// TwinCAT 3 PLC project Untitled1
// ProgramVersion: 3.1.4026.11
// libraries:
//   Tc2_Standard, * (Beckhoff Automation GmbH)
//   Tc2_System, * (Beckhoff Automation GmbH)
//   Tc2_Utilities, * (Beckhoff Automation GmbH)
// project tree:
//   CommandInvoker/ FB_CommandInvoker.TcPOU, I_CommandInvoker.TcIO
//   Command/AxisCommandExample/ FB_AxisCommandFactory.TcPOU (not stored), FB_AxisMoveCommand.TcPOU
//   Command/FlowCommands/ FB_CompositeCommand.TcPOU, FB_FlowCommandFactory.TcPOU, FB_WaitCommand.TcPOU, FB_WaitForConditionCommand.TcPOU
//   Command/ I_Command.TcIO
//   Command/ValveCommandExample/ FB_ValveCommandFactory.TcPOU (not stored), FB_ValveMoveCommand.TcPOU
//   Components/Axis/ FB_Axis.TcPOU (not stored), I_Axis.TcIO (not stored)
//   Components/Valve/ E_ValvePosition.TcDUT, FB_Valve.TcPOU, I_Valve.TcIO
//   General/Datatypes/ Integer.TcDUT (not stored), Positive.TcDUT (not stored), Number.TcDUT
//   General/ FB_Base.TcPOU, F_Log.TcPOU
//   InplaceStringBuilder/ FB_StringBuilder.TcPOU, F_BuildString.TcPOU
//   / MAIN.TcPOU, PlcTask.TcTTO
//   Progress/ E_ProgressStatus.TcDUT, FB_Progress.TcPOU, I_Progress.TcIO
//   Values/Binding/ Value.TcPOU, FB_BoolBindingReadOnly.TcPOU, I_BoolBindable.TcIO (not stored), NotValue.TcPOU
//   Values/BooleanExpression/ Or2.TcPOU, And3.TcPOU, Or3.TcPOU, And4.TcPOU, Or4.TcPOU, And5.TcPOU, Or5.TcPOU, E_BooleanOperator.TcDUT, FB_BooleanExpression.TcPOU, And2.TcPOU
//   Values/ BoolValues.TcGVL, FB_TrueBoolValue.TcPOU, FB_FalseBoolValue.TcPOU, I_BoolValue.TcIO
// real-time tasks:
//   TASK PlcTask: cycle T#10ms, priority 20, ADS port 350

CONFIGURATION Untitled1
    RESOURCE PLC ON TwinCAT3
        TASK PlcTask(INTERVAL := T#10ms, PRIORITY := 20);
        PROGRAM MAIN WITH PlcTask : MAIN;
    END_RESOURCE
END_CONFIGURATION

// ---- Components/Valve/E_ValvePosition.TcDUT
{attribute 'qualified_only'}
{attribute 'strict'}
{attribute 'to_string'}
TYPE E_ValvePosition :
(
	Home,
	Work
);
END_TYPE

// ---- General/Datatypes/Number.TcDUT
TYPE Number : LREAL; END_TYPE

// ---- Progress/E_ProgressStatus.TcDUT
{attribute 'qualified_only'}
{attribute 'strict'}
{attribute 'to_string'}
TYPE E_ProgressStatus :
(
	Idle,
	Running,
	Paused,
	Completed,
	Error
);
END_TYPE

// ---- Values/BooleanExpression/E_BooleanOperator.TcDUT
{attribute 'qualified_only'}
{attribute 'strict'}
{attribute 'to_string'}
TYPE E_BooleanOperator :
(
	ANDop,
	ORop,
	XORop
);
END_TYPE

// ---- Values/BoolValues.TcGVL
{attribute 'qualified_only'}
VAR_GLOBAL CONSTANT
	FalseValue : FB_FalseBoolValue := ();
	TrueValue : FB_TrueBoolValue := ();
END_VAR

// ---- CommandInvoker/I_CommandInvoker.TcIO
INTERFACE I_CommandInvoker

METHOD AddCommand : BOOL
VAR_INPUT
	command : I_Command;
END_VAR
END_METHOD

METHOD ClearCommands
VAR
END_VAR
END_METHOD

{attribute 'monitoring' := 'call'}
PROPERTY CommandCount : INT
GET
END_GET
END_PROPERTY

METHOD Cyclic
VAR_INPUT
END_VAR
END_METHOD

{attribute 'monitoring' := 'call'}
PROPERTY InvokeIndex : INT
GET
END_GET
END_PROPERTY

METHOD Pause
VAR_INPUT
END_VAR
END_METHOD

{attribute 'monitoring' := 'call'}
PROPERTY PauseRequest : BOOL
GET
END_GET
END_PROPERTY

{attribute 'monitoring' := 'call'}
PROPERTY ProgressPercent : REAL
GET
END_GET
END_PROPERTY

{attribute 'monitoring' := 'call'}
PROPERTY ProgressState : E_ProgressStatus
GET
END_GET
END_PROPERTY

METHOD Reset
VAR_INPUT
END_VAR
END_METHOD

METHOD ResetCommands : BOOL
VAR
END_VAR
END_METHOD

METHOD Start
VAR_INPUT
END_VAR
END_METHOD

{attribute 'monitoring' := 'call'}
PROPERTY StepMode : BOOL
GET
END_GET
SET
END_SET
END_PROPERTY

END_INTERFACE

// ---- Command/I_Command.TcIO
INTERFACE I_Command EXTENDS __SYSTEM.IQueryInterface

{attribute 'monitoring' := 'call'}
PROPERTY Description : STRING
GET
END_GET
END_PROPERTY

METHOD Execute : E_ProgressStatus
VAR_INPUT
END_VAR
END_METHOD

METHOD Reset
VAR_INPUT
END_VAR
END_METHOD

END_INTERFACE

// ---- Components/Valve/I_Valve.TcIO
INTERFACE I_Valve

METHOD MoveToHome : BOOL
VAR_INPUT
END_VAR
END_METHOD

METHOD MoveToWork : BOOL
VAR_INPUT
END_VAR
END_METHOD

END_INTERFACE

// ---- Progress/I_Progress.TcIO
INTERFACE I_Progress

{attribute 'monitoring' := 'call'}
PROPERTY CompletedCount : INT
GET
END_GET
SET
END_SET
END_PROPERTY

{attribute 'monitoring' := 'call'}
PROPERTY Count : INT
GET
END_GET
SET
END_SET
END_PROPERTY

{attribute 'monitoring' := 'call'}
PROPERTY Percent : REAL
GET
END_GET
END_PROPERTY

{attribute 'monitoring' := 'call'}
PROPERTY PercentString : STRING
GET
END_GET
END_PROPERTY

{attribute 'monitoring' := 'call'}
PROPERTY UnitProgress : REAL // Progress 0..1
GET
END_GET
END_PROPERTY

END_INTERFACE

// ---- Values/I_BoolValue.TcIO
INTERFACE I_BoolValue EXTENDS __SYSTEM.IQueryInterface

{attribute 'monitoring' := 'call'}
PROPERTY Value : BOOL
GET
END_GET
END_PROPERTY

END_INTERFACE

// ---- MAIN.TcPOU
PROGRAM MAIN
VAR
	valve : FB_Valve;
	axis : FB_Axis;
	valveFactory : FB_ValveCommandFactory;
	axisFactory : FB_AxisCommandFactory;
	flowFactory : FB_FlowCommandFactory;
	
	invoker : FB_CommandInvoker<20>;
	subsequence : FB_CommandInvoker<10>;
	
	start : BOOL;
	create : BOOL;
	
	pauseIndex : INT := -1;
	
	test : BOOL;
	test2 : BOOL;
	test3 : BOOL;
	test4 : BOOL;
	
	val : I_BoolValue;
END_VAR

IF create THEN
	create := FALSE;
	
	subsequence.AddCommand(valveFactory.CreateCommand(valve := valve, target := E_ValvePosition.Home, 'move valve to home'));
	subsequence.AddCommand(axisFactory.CreateCommand(axis := axis, target := 50, 'move axis to position'));
	subsequence.AddCommand(valveFactory.CreateCommand(valve := valve, target := E_ValvePosition.Work, 'move valve to work'));

	// This is replacement for a CASE OF state machines
	invoker.AddCommand(valveFactory.CreateCommand(valve := valve, target := E_ValvePosition.Home, 'move valve to home'));
	invoker.AddCommand(axisFactory.CreateCommand(axis := axis, target := 50, 'move axis to position'));
	invoker.AddCommand(valveFactory.CreateCommand(valve := valve, target := E_ValvePosition.Work, 'move valve to work'));
	invoker.AddCommand(flowFactory.CreateCompositeCommand(invoker := subsequence, 'run subsequence'));
// 	invoker.AddCommand(flowFactory.CreateWaitForConditionCommand(And2(Value(test2), Value(test3)), T#0S, T#0S, 'Wait for test2 AND test3'));
	invoker.AddCommand(axisFactory.CreateCommand(axis := axis, target := 0, 'move axis to away'));
// 	invoker.AddCommand(flowFactory.CreateWaitForConditionCommand(NotValue(test2), T#10S, T#0S, 'Wait at least for NOT test2'));
	invoker.AddCommand(valveFactory.CreateCommand(valve := valve, target := E_ValvePosition.Home, 'move valve to home'));
// 	invoker.AddCommand(flowFactory.CreateWaitForConditionCommand(NotValue(test3), T#0S, T#10S, 'Wait for NOT test3, but maximum 10 seconds'));
	invoker.AddCommand(valveFactory.CreateCommand(valve := valve, target := E_ValvePosition.Work, 'move valve to work'));
	invoker.AddCommand(flowFactory.CreateWaitCommand(T#5S, 'wait some time'));
	invoker.AddCommand(valveFactory.CreateCommand(valve := valve, target := E_ValvePosition.Home, 'move valve to home'));
END_IF

IF start THEN
	start := FALSE;
	
	invoker.Start();
END_IF

invoker.Cyclic();

IF (invoker.InvokeIndex = pauseIndex AND invoker.ProgressState <> E_ProgressStatus.Paused) THEN
	invoker.Pause();
END_IF

IF test THEN
	test := FALSE;
	val := And2(Value(test4), Or2(Value(test2), NotValue(test3)));
END_IF

IF (val <> 0) THEN
	val.Value;
END_IF

END_PROGRAM

// ---- Components/Valve/FB_Valve.TcPOU
FUNCTION_BLOCK FB_Valve EXTENDS FB_Base IMPLEMENTS I_Valve
VAR_INPUT
END_VAR
VAR_OUTPUT
END_VAR
VAR
END_VAR

METHOD MoveToHome : BOOL
VAR_INPUT
END_VAR
Tc2_System.ADSLOGSTR(0, 'valve move to home', '');

MoveToHome := TRUE;
END_METHOD

METHOD MoveToWork : BOOL
VAR_INPUT
END_VAR
Tc2_System.ADSLOGSTR(0, 'valve move to work', '');

MoveToWork := TRUE;
END_METHOD

END_FUNCTION_BLOCK

// ---- General/FB_Base.TcPOU
{attribute 'reflection'}
FUNCTION_BLOCK FB_Base
VAR
    {attribute 'instance-path'} 
    {attribute 'noinit'} 
    _InstanceName : STRING;
END_VAR

{attribute 'monitoring' := 'call'}
PROPERTY InstanceName : STRING
GET
InstanceName := _InstanceName;
END_GET
END_PROPERTY

END_FUNCTION_BLOCK

// ---- Command/FlowCommands/FB_FlowCommandFactory.TcPOU
FUNCTION_BLOCK FB_FlowCommandFactory
VAR
END_VAR

METHOD CreateCompositeCommand : I_Command
VAR_INPUT
	invoker : I_CommandInvoker;
	description : STRING;
END_VAR
VAR	
	point : POINTER TO FB_CompositeCommand;
END_VAR
point := __NEW(FB_CompositeCommand(invoker := invoker, description := description));
CreateCompositeCommand := point^;
END_METHOD

METHOD CreateWaitCommand : I_Command
VAR_INPUT
	waitTime : TIME;
	description : STRING;
END_VAR
VAR	
	point : POINTER TO FB_WaitCommand;
END_VAR
point := __NEW(FB_WaitCommand(waitTime := waitTime, description := description));
CreateWaitCommand := point^;
END_METHOD

METHOD CreateWaitForConditionCommand : I_Command
VAR_INPUT
	condition : I_BoolValue;
	minWaitTime : TIME;
	maxWaitTime : TIME;
	description : STRING;
END_VAR
VAR	
	point : POINTER TO FB_WaitForConditionCommand;
END_VAR
point := __NEW(FB_WaitForConditionCommand(condition := condition, minWaitTime := minWaitTime, maxWaitTime := maxWaitTime, description := description));
CreateWaitForConditionCommand := point^;
END_METHOD

END_FUNCTION_BLOCK

// ---- Command/FlowCommands/FB_CompositeCommand.TcPOU
{attribute 'enable_dynamic_creation'}
FUNCTION_BLOCK FB_CompositeCommand IMPLEMENTS I_Command
VAR
	invoker : I_CommandInvoker;
	_Description : STRING;
	
	started : BOOL;
END_VAR

{attribute 'monitoring' := 'call'}
PROPERTY Description : STRING
GET
Description := _Description;
END_GET
END_PROPERTY

METHOD Execute : E_ProgressStatus
IF (NOT started) THEN
	started := TRUE;
	
	invoker.Reset();
	invoker.Start();
END_IF

invoker.Cyclic();

Execute := invoker.ProgressState;
END_METHOD

//FB_Init is always available implicitly and it is used primarily for initialization.
//The return value is not evaluated. For a specific influence, you can also declare the
//methods explicitly and provide additional code there with the standard initialization
//code. You can evaluate the return value.
METHOD FB_Init: BOOL
VAR_INPUT
    bInitRetains: BOOL; // TRUE: the retain variables are initialized (reset warm / reset cold)
    bInCopyCode: BOOL;  // TRUE: the instance will be copied to the copy code afterward (online change)   
	
	invoker : I_CommandInvoker;
	description : STRING;
END_VAR
THIS^.invoker := invoker;
_Description := description;
END_METHOD

METHOD Reset
VAR_INPUT
END_VAR
started := FALSE;
invoker.Reset();
END_METHOD

END_FUNCTION_BLOCK

// ---- Command/FlowCommands/FB_WaitCommand.TcPOU
{attribute 'enable_dynamic_creation'}
FUNCTION_BLOCK FB_WaitCommand IMPLEMENTS I_Command
VAR
	waitTime : TIME;
	waiter : TON;
	_Description : STRING;
END_VAR

{attribute 'monitoring' := 'call'}
PROPERTY Description : STRING
GET
Description := _Description;
END_GET
END_PROPERTY

METHOD Execute : E_ProgressStatus
waiter(IN := TRUE, PT := waitTime);

IF (waiter.Q) THEN
	Execute := E_ProgressStatus.Completed;
ELSE
	Execute := E_ProgressStatus.Running;
END_IF
END_METHOD

//FB_Init is always available implicitly and it is used primarily for initialization.
//The return value is not evaluated. For a specific influence, you can also declare the
//methods explicitly and provide additional code there with the standard initialization
//code. You can evaluate the return value.
METHOD FB_Init: BOOL
VAR_INPUT
    bInitRetains: BOOL; // TRUE: the retain variables are initialized (reset warm / reset cold)
    bInCopyCode: BOOL;  // TRUE: the instance will be copied to the copy code afterward (online change)   
	
	waitTime : TIME;
	description : STRING;
END_VAR
THIS^.waitTime := waitTime;
_Description := description;
END_METHOD

METHOD Reset
VAR_INPUT
END_VAR
waiter(IN := FALSE);
END_METHOD

END_FUNCTION_BLOCK

// ---- Command/FlowCommands/FB_WaitForConditionCommand.TcPOU
{attribute 'enable_dynamic_creation'}
FUNCTION_BLOCK FB_WaitForConditionCommand IMPLEMENTS I_Command
VAR
	condition : I_BoolValue;
	minWaitTime : TIME;
	maxWaitTime : TIME;
	minWaiter : TON;
	maxWaiter : TON;
	_Description : STRING;
END_VAR

{attribute 'monitoring' := 'call'}
PROPERTY Description : STRING
GET
Description := _Description;
END_GET
END_PROPERTY

METHOD Execute : E_ProgressStatus
minWaiter(IN := TRUE, PT := minWaitTime);
maxWaiter(IN := maxWaitTime > T#0S, PT := maxWaitTime);

IF ((condition.Value AND minWaiter.Q) OR maxWaiter.Q) THEN
	Execute := E_ProgressStatus.Completed;
ELSE
	Execute := E_ProgressStatus.Running;
END_IF
END_METHOD

//FB_Init is always available implicitly and it is used primarily for initialization.
//The return value is not evaluated. For a specific influence, you can also declare the
//methods explicitly and provide additional code there with the standard initialization
//code. You can evaluate the return value.
METHOD FB_Init: BOOL
VAR_INPUT
    bInitRetains: BOOL; // TRUE: the retain variables are initialized (reset warm / reset cold)
    bInCopyCode: BOOL;  // TRUE: the instance will be copied to the copy code afterward (online change)   
	
	condition : I_BoolValue;
	minWaitTime : TIME;
	maxWaitTime : TIME;
	description : STRING;
END_VAR
THIS^.condition := condition;
THIS^.minWaitTime := minWaitTime;
THIS^.maxWaitTime := maxWaitTime;
_Description := description;
END_METHOD

METHOD Reset
VAR_INPUT
END_VAR
minWaiter(IN := FALSE);
maxWaiter(IN := FALSE);
END_METHOD

END_FUNCTION_BLOCK

// ---- Values/Binding/Value.TcPOU
FUNCTION Value : I_BoolValue
VAR_INPUT
	boolean : REFERENCE TO BOOL;
END_VAR
VAR
	p : POINTER TO FB_BoolBindingReadOnly;
END_VAR

p := __NEW(FB_BoolBindingReadOnly);

p^.Bind(boolean);

Value := p^;

END_FUNCTION

// ---- Values/Binding/FB_BoolBindingReadOnly.TcPOU
{attribute 'enable_dynamic_creation'}
FUNCTION_BLOCK FB_BoolBindingReadOnly IMPLEMENTS I_BoolBindable
VAR
	ref : REFERENCE TO BOOL;
	_Negate : BOOL;
END_VAR

METHOD Bind
VAR_INPUT
	boolean : REFERENCE TO BOOL;
END_VAR
ref REF= boolean;
END_METHOD

{attribute 'monitoring' := 'call'}
PROPERTY IsBinded : BOOL
GET
IsBinded := __ISVALIDREF(ref);
END_GET
END_PROPERTY

PROPERTY Negate : BOOL
GET
Negate := _Negate;
END_GET
SET
_Negate := Negate;
END_SET
END_PROPERTY

{attribute 'monitoring' := 'call'}
PROPERTY Value : BOOL
GET
Value := ref XOR _Negate;
END_GET
END_PROPERTY

END_FUNCTION_BLOCK

// ---- CommandInvoker/FB_CommandInvoker.TcPOU
FUNCTION_BLOCK FB_CommandInvoker
VAR_GENERIC CONSTANT
	CommandCapacity : INT := 10;
END_VAR
EXTENDS FB_Base IMPLEMENTS I_CommandInvoker
VAR
	_Commands : ARRAY[0..CommandCapacity - 1] OF I_Command;
	_CommandCount : INT;
	
	_InvokeIndex : INT;
	_ProgressState : E_ProgressStatus;
	
	_PauseRequest : BOOL;
	_StepMode : BOOL;
END_VAR

METHOD AddCommand : BOOL
VAR_INPUT
	command : I_Command;
END_VAR
IF (NOT _CommandCount < CommandCapacity) THEN
	F_Log('Can not add any more commands!');
	RETURN;
END_IF

_Commands[_CommandCount] := command;
_CommandCount := _CommandCount + 1;

AddCommand := TRUE;
END_METHOD

METHOD ClearCommands
VAR
	i : INT;
	p : POINTER TO BYTE;
END_VAR
FOR i := 0 TO _CommandCount - 1 DO
	__QUERYPOINTER(_Commands[i], p);
	__DELETE(p);
END_FOR

_CommandCount := 0;
END_METHOD

{attribute 'monitoring' := 'call'}
PROPERTY CommandCount : INT
GET
CommandCount := _CommandCount;
END_GET
END_PROPERTY

{attribute 'monitoring' := 'call'}
PROPERTY Commands : REFERENCE TO ARRAY[0..CommandCapacity - 1] OF I_Command
GET
Commands REF= _Commands;
END_GET
END_PROPERTY

METHOD Cyclic
VAR_INPUT
END_VAR
IF (_ProgressState = E_ProgressStatus.Running) THEN
	Invoke();
END_IF
END_METHOD

//FB_Exit must be implemented explicitly. If there is an implementation, then the
//method is called before the controller removes the code of the function block instance
//(implicit call). The return value is not evaluated.
METHOD FB_Exit: BOOL
VAR_INPUT
    bInCopyCode: BOOL;  // TRUE: the exit method is called in order to leave the instance which will be copied afterwards (online change).  
END_VAR
ClearCommands();
END_METHOD

METHOD PRIVATE Invoke
VAR
	commandProgress : E_ProgressStatus;
	progress : T_MaxString;
	test : STRING := 'test';
END_VAR
IF (_CommandCount = 0) THEN
	_ProgressState := E_ProgressStatus.Completed;
	
	F_Log('Invoker finished. No commands were executed.');	
END_IF

IF (_InvokeIndex < _CommandCount) THEN
	
	commandProgress := _Commands[_InvokeIndex].Execute();
	IF (commandProgress = E_ProgressStatus.Completed) THEN
		
		F_Log(F_BuildString('Command "').Append(_Commands[_InvokeIndex].Description).Append('" has finished!').GetString());
		
		IF (_PauseRequest OR _StepMode) THEN
			_ProgressState := E_ProgressStatus.Paused;
			_PauseRequest := FALSE;
		END_IF
		
		IF (_InvokeIndex = _CommandCount - 1) THEN
			_ProgressState := E_ProgressStatus.Completed;
			
			F_Log('Invoker finished');
		END_IF

		_InvokeIndex := _InvokeIndex + 1;
		
		F_Log(
			F_BuildString('Invoker progress  ')
				.Append(TO_STRING(_InvokeIndex))
				.Append('/')
				.Append(TO_STRING(_CommandCount))
				.Append('  ')
				.Append(LREAL_TO_FMTSTR(ProgressPercent, 1, TRUE))
				.Append(' %s')
				.GetString());
	END_IF
END_IF
END_METHOD

{attribute 'monitoring' := 'call'}
PROPERTY InvokeIndex : INT
GET
InvokeIndex := _InvokeIndex;
END_GET
END_PROPERTY

METHOD Pause
VAR_INPUT
END_VAR
_PauseRequest := TRUE;
END_METHOD

{attribute 'monitoring' := 'call'}
PROPERTY PauseRequest : BOOL
GET
PauseRequest := _PauseRequest;
END_GET
END_PROPERTY

{attribute 'monitoring' := 'call'}
PROPERTY ProgressPercent : REAL
GET
IF (_CommandCount > 0) THEN
	ProgressPercent := 100.0 * _InvokeIndex / _CommandCount;
ELSE
	ProgressPercent := 0;
END_IF
END_GET
END_PROPERTY

{attribute 'monitoring' := 'call'}
PROPERTY ProgressState : E_ProgressStatus
GET
ProgressState := _ProgressState;
END_GET
END_PROPERTY

METHOD Reset
VAR_INPUT
END_VAR
_InvokeIndex := 0;
_ProgressState := E_ProgressStatus.Idle;

_PauseRequest := FALSE;

ResetCommands();
END_METHOD

METHOD ResetCommands : BOOL
VAR
	i : INT;
END_VAR
FOR i := 0 TO _CommandCount - 1 DO
	_Commands[i].Reset();
END_FOR
END_METHOD

METHOD Start
VAR_INPUT
END_VAR
CASE _ProgressState OF
	
	E_ProgressStatus.Idle,
	E_ProgressStatus.Paused,
	E_ProgressStatus.Completed:
		
		IF (NOT(_ProgressState = E_ProgressStatus.Paused
				OR (_ProgressState = E_ProgressStatus.Running AND (_PauseRequest OR _StepMode)))) THEN
			
			_InvokeIndex := 0;
			
			ResetCommands();
		END_IF
		
		_ProgressState := E_ProgressStatus.Running;
		_PauseRequest := FALSE;

		F_Log('Invoker started');
END_CASE
END_METHOD

{attribute 'monitoring' := 'call'}
PROPERTY StepMode : BOOL
GET
StepMode := _StepMode;
END_GET
SET
_StepMode := StepMode;
END_SET
END_PROPERTY

END_FUNCTION_BLOCK

// ---- General/F_Log.TcPOU
FUNCTION F_Log
VAR_INPUT
	value : T_MaxString;
END_VAR

Tc2_System.ADSLOGSTR(0, value, '%');

END_FUNCTION

// ---- InplaceStringBuilder/F_BuildString.TcPOU
FUNCTION F_BuildString : REFERENCE TO FB_StringBuilder
VAR_INPUT
	value : T_MaxString;
END_VAR
VAR
END_VAR
VAR_STAT
	builder : FB_StringBuilder;
END_VAR

builder.Clear();

builder.Append(value);

F_BuildString REF= builder;

END_FUNCTION

// ---- InplaceStringBuilder/FB_StringBuilder.TcPOU
FUNCTION_BLOCK FB_StringBuilder
VAR
	_value : T_MaxString;
END_VAR

METHOD Append : REFERENCE TO FB_StringBuilder
VAR_INPUT
	value : T_MaxString;
END_VAR
_value := CONCAT(_value, value);

Append REF= THIS^;
END_METHOD

METHOD Clear : REFERENCE TO FB_StringBuilder
VAR_INPUT
END_VAR
_value := '';

Clear REF= THIS^;
END_METHOD

METHOD GetString : T_MaxString
VAR_INPUT
END_VAR
GetString := _value;
END_METHOD

END_FUNCTION_BLOCK

// ---- Values/BooleanExpression/And2.TcPOU
FUNCTION And2 : I_BoolValue
VAR_INPUT
	value1 : I_BoolValue;
	value2 : I_BoolValue;
END_VAR
VAR
	p : POINTER TO FB_BooleanExpression;
END_VAR

p := __NEW(FB_BooleanExpression);

p^.Op2(
	operator := E_BooleanOperator.ANDop,
	value1 := value1,
	value2 := value2
);

And2 := p^;

END_FUNCTION

// ---- Values/BooleanExpression/FB_BooleanExpression.TcPOU
{attribute 'enable_dynamic_creation'}
FUNCTION_BLOCK FB_BooleanExpression IMPLEMENTS I_BoolValue
VAR
	operands : ARRAY[0..MaxBooleanExpressionOperandCount - 1] OF I_BoolValue;
	operandCount : INT;
	operator : E_BooleanOperator;
END_VAR
VAR CONSTANT
	MaxBooleanExpressionOperandCount : INT := 5;
END_VAR

METHOD Clear
VAR
	i : INT;
	p : POINTER TO BYTE;
END_VAR
FOR i := 0 TO operandCount - 1 DO
	__QUERYPOINTER(operands[i], p);
	__DELETE(p);
	operands[i] := 0;
END_FOR

operandCount := 0;
END_METHOD

METHOD Op2
VAR_INPUT
	operator : E_BooleanOperator;
	value1 : I_BoolValue;
	value2 : I_BoolValue;
END_VAR
Clear();

THIS^.operator := operator;

operands[0] := value1;
operands[1] := value2;
operandCount := 2;
END_METHOD

METHOD Op3
VAR_INPUT
	operator : E_BooleanOperator;
	value1 : I_BoolValue;
	value2 : I_BoolValue;
	value3 : I_BoolValue;
END_VAR
Clear();

THIS^.operator := operator;

operands[0] := value1;
operands[1] := value2;
operands[2] := value3;
operandCount := 3;
END_METHOD

METHOD Op4
VAR_INPUT
	operator : E_BooleanOperator;
	value1 : I_BoolValue;
	value2 : I_BoolValue;
	value3 : I_BoolValue;
	value4 : I_BoolValue;
END_VAR
Clear();

THIS^.operator := operator;

operands[0] := value1;
operands[1] := value2;
operands[2] := value3;
operands[3] := value4;
operandCount := 4;
END_METHOD

METHOD Op5
VAR_INPUT
	operator : E_BooleanOperator;
	value1 : I_BoolValue;
	value2 : I_BoolValue;
	value3 : I_BoolValue;
	value4 : I_BoolValue;
	value5 : I_BoolValue;
END_VAR
Clear();

THIS^.operator := operator;

operands[0] := value1;
operands[1] := value2;
operands[2] := value3;
operands[3] := value4;
operands[4] := value5;
operandCount := 5;
END_METHOD

{attribute 'monitoring' := 'call'}
PROPERTY Value : BOOL
GET
VAR
	i : INT;
	result : BOOL;
END_VAR
IF (operandCount = 0) THEN
	RETURN;
END_IF

CASE operator OF
	
	E_BooleanOperator.ANDop:
		
		result := operands[0].Value;
		FOR i := 1 TO operandCount - 1 DO
			result := result AND operands[i].Value;
		END_FOR	
		
	E_BooleanOperator.ORop:
		
		result := operands[0].Value;
		FOR i := 1 TO operandCount - 1 DO
			result := result OR operands[i].Value;
		END_FOR	
		
	E_BooleanOperator.XORop:
		
		result := operands[0].Value;
		FOR i := 1 TO operandCount - 1 DO
			result := result XOR operands[i].Value;
		END_FOR	
		
END_CASE

Value := result;
END_GET
END_PROPERTY

END_FUNCTION_BLOCK

// ---- Values/BooleanExpression/Or2.TcPOU
FUNCTION Or2 : I_BoolValue
VAR_INPUT
	value1 : I_BoolValue;
	value2 : I_BoolValue;
END_VAR
VAR
	p : POINTER TO FB_BooleanExpression;
END_VAR

p := __NEW(FB_BooleanExpression);

p^.Op2(
	operator := E_BooleanOperator.ORop,
	value1 := value1,
	value2 := value2
);

Or2 := p^;

END_FUNCTION

// ---- Values/Binding/NotValue.TcPOU
FUNCTION NotValue : I_BoolValue
VAR_INPUT
	boolean : REFERENCE TO BOOL;
END_VAR
VAR
	p : POINTER TO FB_BoolBindingReadOnly;
END_VAR

p := __NEW(FB_BoolBindingReadOnly);

p^.Bind(boolean);
p^.Negate := TRUE;

NotValue := p^;

END_FUNCTION

// ---- Values/FB_FalseBoolValue.TcPOU
FUNCTION_BLOCK FB_FalseBoolValue IMPLEMENTS I_BoolValue
VAR
END_VAR

{attribute 'monitoring' := 'call'}
PROPERTY Value : BOOL
GET
Value := FALSE;
END_GET
END_PROPERTY

END_FUNCTION_BLOCK

// ---- Values/FB_TrueBoolValue.TcPOU
FUNCTION_BLOCK FB_TrueBoolValue IMPLEMENTS I_BoolValue
VAR
END_VAR

{attribute 'monitoring' := 'call'}
PROPERTY Value : BOOL
GET
Value := TRUE;
END_GET
END_PROPERTY

END_FUNCTION_BLOCK

// ---- Command/AxisCommandExample/FB_AxisMoveCommand.TcPOU
{attribute 'enable_dynamic_creation'}
FUNCTION_BLOCK FB_AxisMoveCommand IMPLEMENTS I_Command
VAR
	_Axis : I_Axis;
	_Target : REAL;
	_Description : STRING;
END_VAR

{attribute 'monitoring' := 'call'}
PROPERTY Description : STRING
GET
Description := _Description;
END_GET
END_PROPERTY

METHOD Execute : E_Progress
_Axis.MoveAbsolute(_target);

Execute := E_Progress.Completed;
END_METHOD

//FB_Init is always available implicitly and it is used primarily for initialization.
//The return value is not evaluated. For a specific influence, you can also declare the
//methods explicitly and provide additional code there with the standard initialization
//code. You can evaluate the return value.
METHOD FB_Init: BOOL
VAR_INPUT
    bInitRetains: BOOL; // TRUE: the retain variables are initialized (reset warm / reset cold)
    bInCopyCode: BOOL;  // TRUE: the instance will be copied to the copy code afterward (online change)   
	
	axis : I_Axis;
	target : REAL;
	description : STRING;
END_VAR
_Axis := axis;
_Target := target;
_Description := description;
END_METHOD

METHOD Reset
VAR_INPUT
END_VAR
// nothing to reset here
END_METHOD

END_FUNCTION_BLOCK

// ---- Command/ValveCommandExample/FB_ValveMoveCommand.TcPOU
{attribute 'enable_dynamic_creation'}
FUNCTION_BLOCK FB_ValveMoveCommand IMPLEMENTS I_Command
VAR
	_Valve : I_Valve;
	_Target : E_ValvePosition;
	_Description : STRING;
END_VAR

{attribute 'monitoring' := 'call'}
PROPERTY Description : STRING
GET
Description := _Description;
END_GET
END_PROPERTY

METHOD Execute : E_ProgressStatus
CASE _Target OF
	
	E_ValvePosition.Home:
		_Valve.MoveToHome();
	
	E_ValvePosition.Work:
		_Valve.MoveToWork();
END_CASE

Execute := E_ProgressStatus.Completed;
END_METHOD

//FB_Init is always available implicitly and it is used primarily for initialization.
//The return value is not evaluated. For a specific influence, you can also declare the
//methods explicitly and provide additional code there with the standard initialization
//code. You can evaluate the return value.
METHOD FB_Init: BOOL
VAR_INPUT
    bInitRetains: BOOL; // TRUE: the retain variables are initialized (reset warm / reset cold)
    bInCopyCode: BOOL;  // TRUE: the instance will be copied to the copy code afterward (online change)   
	
	valve : I_Valve;
	target : E_ValvePosition;
	description : STRING;
END_VAR
_Valve := valve;
_Target := target;
_Description := description;
END_METHOD

METHOD Reset
VAR_INPUT
END_VAR
// nothing to reset here
END_METHOD

END_FUNCTION_BLOCK

// ---- Progress/FB_Progress.TcPOU
FUNCTION_BLOCK FB_Progress IMPLEMENTS I_Progress
VAR
	_Count : INT;
	_CompletedCount : INT;
	
	_ParentProgress : I_Progress;
END_VAR

{attribute 'monitoring' := 'call'}
PROPERTY CompletedCount : INT
GET
CompletedCount := _CompletedCount;
END_GET
SET
_CompletedCount := CompletedCount;
END_SET
END_PROPERTY

{attribute 'monitoring' := 'call'}
PROPERTY Count : INT
GET
Count := _Count;
END_GET
SET
_Count := Count;
END_SET
END_PROPERTY

{attribute 'monitoring' := 'call'}
PROPERTY Percent : REAL
GET
Percent := 100.0 * UnitProgress;
END_GET
END_PROPERTY

{attribute 'monitoring' := 'call'}
PROPERTY PercentString : STRING
GET
PercentString := CONCAT(LREAL_TO_FMTSTR(Percent, 1, TRUE), ' %');
END_GET
END_PROPERTY

{attribute 'monitoring' := 'call'}
PROPERTY UnitProgress : REAL // Progress 0..1
GET
IF (_Count = 0) THEN
	UnitProgress := 0;
	RETURN;
END_IF

UnitProgress := _CompletedCount / _Count;
END_GET
END_PROPERTY

END_FUNCTION_BLOCK

// ---- Values/BooleanExpression/And3.TcPOU
FUNCTION And3 : I_BoolValue
VAR_INPUT
	value1 : I_BoolValue;
	value2 : I_BoolValue;
	value3 : I_BoolValue;
END_VAR
VAR
	p : POINTER TO FB_BooleanExpression;
END_VAR

p := __NEW(FB_BooleanExpression);

p^.Op3(
	operator := E_BooleanOperator.ANDop,
	value1 := value1,
	value2 := value2,
	value3 := value3
);

And3 := p^;

END_FUNCTION

// ---- Values/BooleanExpression/Or3.TcPOU
FUNCTION Or3 : I_BoolValue
VAR_INPUT
	value1 : I_BoolValue;
	value2 : I_BoolValue;
	value3 : I_BoolValue;
END_VAR
VAR
	p : POINTER TO FB_BooleanExpression;
END_VAR

p := __NEW(FB_BooleanExpression);

p^.Op3(
	operator := E_BooleanOperator.ORop,
	value1 := value1,
	value2 := value2,
	value3 := value3
);

Or3 := p^;

END_FUNCTION

// ---- Values/BooleanExpression/And4.TcPOU
FUNCTION And4 : I_BoolValue
VAR_INPUT
	value1 : I_BoolValue;
	value2 : I_BoolValue;
	value3 : I_BoolValue;
	value4 : I_BoolValue;
END_VAR
VAR
	p : POINTER TO FB_BooleanExpression;
END_VAR

p := __NEW(FB_BooleanExpression);

p^.Op4(
	operator := E_BooleanOperator.ANDop,
	value1 := value1,
	value2 := value2,
	value3 := value3,
	value4 := value4
);

And4 := p^;

END_FUNCTION

// ---- Values/BooleanExpression/Or4.TcPOU
FUNCTION Or4 : I_BoolValue
VAR_INPUT
	value1 : I_BoolValue;
	value2 : I_BoolValue;
	value3 : I_BoolValue;
	value4 : I_BoolValue;
END_VAR
VAR
	p : POINTER TO FB_BooleanExpression;
END_VAR

p := __NEW(FB_BooleanExpression);

p^.Op4(
	operator := E_BooleanOperator.ORop,
	value1 := value1,
	value2 := value2,
	value3 := value3,
	value4 := value4
);

Or4 := p^;

END_FUNCTION

// ---- Values/BooleanExpression/And5.TcPOU
FUNCTION And5 : I_BoolValue
VAR_INPUT
	value1 : I_BoolValue;
	value2 : I_BoolValue;
	value3 : I_BoolValue;
	value4 : I_BoolValue;
	value5 : I_BoolValue;
END_VAR
VAR
	p : POINTER TO FB_BooleanExpression;
END_VAR

p := __NEW(FB_BooleanExpression);

p^.Op5(
	operator := E_BooleanOperator.ANDop,
	value1 := value1,
	value2 := value2,
	value3 := value3,
	value4 := value4,
	value5 := value5
);

And5 := p^;

END_FUNCTION

// ---- Values/BooleanExpression/Or5.TcPOU
FUNCTION Or5 : I_BoolValue
VAR_INPUT
	value1 : I_BoolValue;
	value2 : I_BoolValue;
	value3 : I_BoolValue;
	value4 : I_BoolValue;
	value5 : I_BoolValue;
END_VAR
VAR
	p : POINTER TO FB_BooleanExpression;
END_VAR

p := __NEW(FB_BooleanExpression);

p^.Op5(
	operator := E_BooleanOperator.ORop,
	value1 := value1,
	value2 := value2,
	value3 := value3,
	value4 := value4,
	value5 := value5
);

Or5 := p^;

END_FUNCTION
